// TIA Portal project "boDem" (V14)

(* hardware
DEVICE "S7-1200 station_1"  S7-1200 Station
   slot 0: "Rack_0"  S7-1200 Rack  Rack  V1.0
   slot 1: "PLC_1"  CPU 1214C DC/DC/DC  6ES7 214-1AG40-0XB0  V4.2
*)

// ===== PLC "PLC_1"  CPU 1214C DC/DC/DC =====

VAR_GLOBAL   // PLC tag table "Default tag table"
   "Tag_1" AT %I0.1 : Bool;
   "Tag_2" AT %I0.3 : Bool;
   "Tag_3" AT %I0.0 : Bool;
   "Tag_4" AT %Q0.2 : Bool;
   "Tag_5" AT %Q0.0 : Bool;
   "Tag_6" AT %Q0.1 : Bool;
END_VAR

// folder: System blocks/Program resources

DATA_BLOCK "t01"   // DB1
{ S7_Optimized_Access := 'TRUE' }
AUTHOR : Simatic
FAMILY : IEC
NAME : IEC_TMR
VERSION : 1.0
// stored: InstanceOfName IEC_TIMER
"IEC_TIMER"
BEGIN
END_DATA_BLOCK

DATA_BLOCK "IEC_Timer_0_DB"   // DB2
{ S7_Optimized_Access := 'TRUE' }
AUTHOR : Simatic
FAMILY : IEC
NAME : IEC_TMR
VERSION : 1.0
// stored: InstanceOfName IEC_TIMER
"IEC_TIMER"
BEGIN
END_DATA_BLOCK

DATA_BLOCK "IEC_Counter_0_DB"   // DB3
{ S7_Optimized_Access := 'TRUE' }
AUTHOR : Simatic
FAMILY : IEC
NAME : CNTR
VERSION : 1.0
// stored: InstanceOfName IEC_COUNTER
"IEC_COUNTER"
BEGIN
END_DATA_BLOCK

// folder: (top level)

ORGANIZATION_BLOCK "Main"   // OB1, LAD, ProgramCycle
TITLE = "Main Program Sweep (Cycle)"
{ S7_Optimized_Access := 'TRUE' }
VERSION : 0.1
   VAR_INPUT
      Initial_Call : Bool;   // Initial call of this OB
      Remanence : Bool;   // =True, if remanent data are available
   END_VAR
BEGIN

REGION Network 1
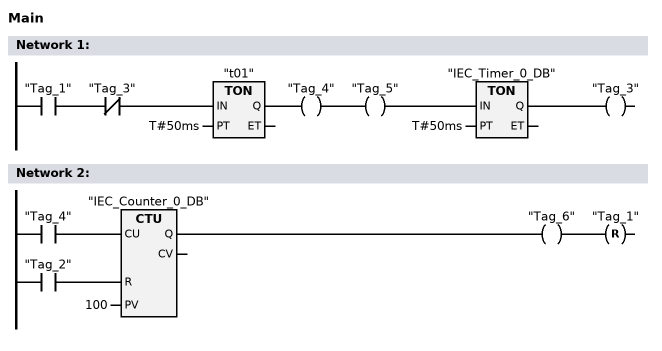
   "t01".TON(IN := "Tag_1" AND NOT "Tag_3", PT := T#50ms);
   "Tag_4" := "t01".Q;
   "Tag_5" := "t01".Q;
   "IEC_Timer_0_DB".TON(IN := "t01".Q, PT := T#50ms);
   "Tag_3" := "IEC_Timer_0_DB".Q;
END_REGION

REGION Network 2
   "IEC_Counter_0_DB".CTU(CU := "Tag_4", R := "Tag_2", PV := 100);
   "Tag_6" := "IEC_Counter_0_DB".Q;
   IF "IEC_Counter_0_DB".Q THEN "Tag_1" := FALSE; END_IF;
END_REGION
END_ORGANIZATION_BLOCK